PROGRAM FILE_BLOCK_DEMO
VAR
	PT : NETWORK_BUFFER;
	fsd : FILE_SERVER_DATA;
	FILE_SERVER : FILE_SERVER;
	FILE_BLOCK : FILE_BLOCK;
	filename : STRING := 'config.ini';
	data : BYTE;
	error : BYTE;
	mode : BYTE;
	pos : UDINT;
END_VAR

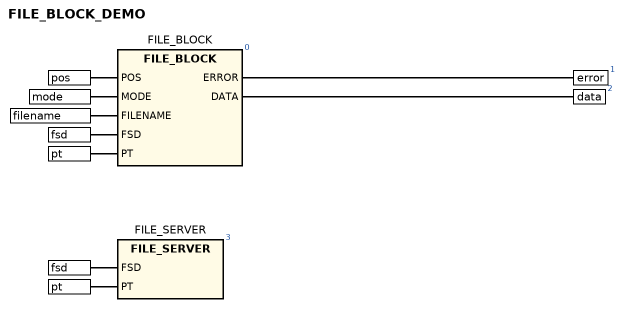
FILE_BLOCK(POS := pos, MODE := mode, FILENAME := filename, FSD := fsd, PT := pt);
error := FILE_BLOCK.ERROR;
data := FILE_BLOCK.DATA;
FILE_SERVER(FSD := fsd, PT := pt);

END_PROGRAM

(* stored: Version 1.1.0.1, ProductVersion 3.1.4024.9
   POU FILE_BLOCK_DEMO: Id {e09d0696-a703-4d3e-9aea-c5d9b567e596}, SpecialFunc None *)
